FUNCTION_BLOCK Test_TExecutionWhenBusy_Abort_SelectsAborting EXTENDS TUnitTestbase
VAR
    Execution : TExecution;
END_VAR

// Setup...
Execution.FB_init(
    bInitRetains := FALSE,
    bInCopyCode  := FALSE);

// Test...
Execution.Start();
Execution.SetBusy();
Execution.Abort();

Assertion.AssertEquals_BOOL(
    Expected := TRUE,
    Actual   := Execution.Aborting,
    VariableName  := 'Execution.Aborting');

TestFinished();

END_FUNCTION_BLOCK

(* stored: Version 1.1.0.1, ProductVersion 3.1.4024.4
   POU Test_TExecutionWhenBusy_Abort_SelectsAborting: Id {81e5767e-c224-40f8-b246-cbf43c4ac2ac}, SpecialFunc None *)
